// TIA Portal V20 export
TYPE "LER_SignalsInterface"
// stored: Access Published
   STRUCT
      HMI_Select_Mode : Bool;
      ButtonValue : Array[0..16] of "LER_SignalsInput";
   END_STRUCT;
END_TYPE
